FUNCTION makeTupleStruct_2: TupleStruct_2
VAR_INPUT
    field0: TupleStruct_1;
    field1: LREAL;
END_VAR
VAR
    rslt: TupleStruct_2;
END_VAR


        rslt.field0 := field0;
rslt.field1 := field1;
makeTupleStruct_2 := rslt;

END_FUNCTION

(* stored: ProductVersion 3.1.0.18, Version 1.1.0.1 *)
